TYPE ST_ItemPK3_OUT1 :
STRUCT
	Identity		:ST_Identity_PK3_OUT1;
	ItemState		:STRING;
	RejectReason	:ST_RejectReason_PK3_OUT1;
	logs			:ST_logs_PK3_OUT1;
	NoRead			:STRING;
END_STRUCT
END_TYPE

(* stored: Version 1.1.0.1, ProductVersion 3.1.4024.13
   DUT ST_ItemPK3_OUT1: Id {5886f7ef-0567-469e-ba84-9b69619877b9} *)
